PROGRAM PRG_11_AirFlowAnalytics
VAR
	AirFlowRateSensor: GenericSensor;
	AirPressureSensor: GenericSensor;
	AirTemperatureSensor: GenericSensor;
	
	AirFlowSensorPublishMqtt: PublishJsonMqtt;
	AirPresSensorPublishMqtt: PublishJsonMqtt;
	AirTempSensorPublishMqtt: PublishJsonMqtt;
END_VAR

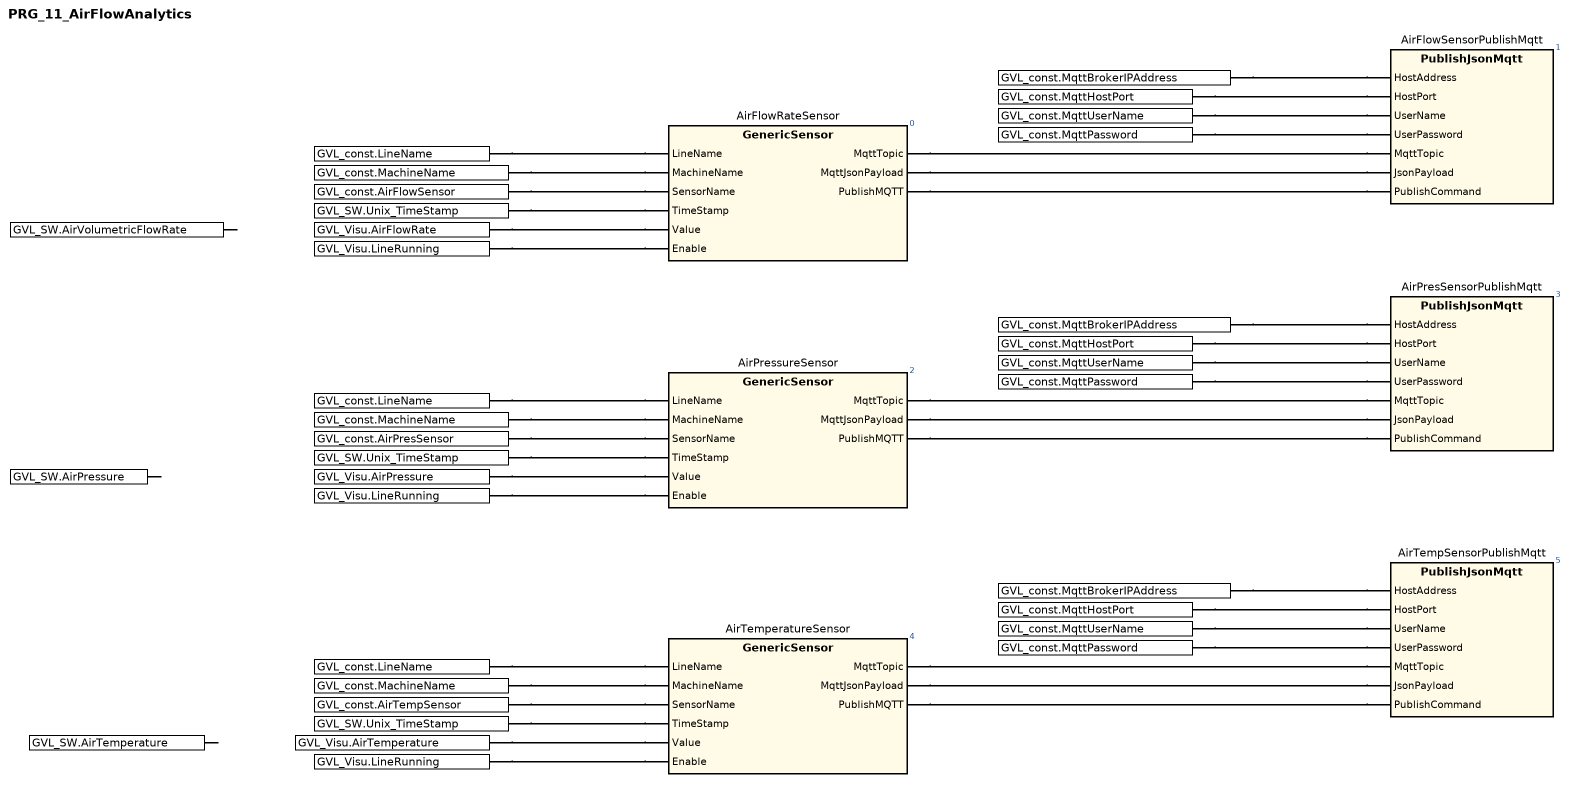
AirFlowRateSensor(
    LineName := GVL_const.LineName,
    MachineName := GVL_const.MachineName,
    SensorName := GVL_const.AirFlowSensor,
    TimeStamp := GVL_SW.Unix_TimeStamp,
    Value := GVL_Visu.AirFlowRate,
    Enable := GVL_Visu.LineRunning); // GenericSensor
AirFlowSensorPublishMqtt(
    HostAddress := GVL_const.MqttBrokerIPAddress,
    HostPort := GVL_const.MqttHostPort,
    UserName := GVL_const.MqttUserName,
    UserPassword := GVL_const.MqttPassword,
    MqttTopic := AirFlowRateSensor.MqttTopic,
    JsonPayload := AirFlowRateSensor.MqttJsonPayload,
    PublishCommand := AirFlowRateSensor.PublishMQTT); // PublishJsonMqtt
AirPressureSensor(
    LineName := GVL_const.LineName,
    MachineName := GVL_const.MachineName,
    SensorName := GVL_const.AirPresSensor,
    TimeStamp := GVL_SW.Unix_TimeStamp,
    Value := GVL_Visu.AirPressure,
    Enable := GVL_Visu.LineRunning); // GenericSensor
AirPresSensorPublishMqtt(
    HostAddress := GVL_const.MqttBrokerIPAddress,
    HostPort := GVL_const.MqttHostPort,
    UserName := GVL_const.MqttUserName,
    UserPassword := GVL_const.MqttPassword,
    MqttTopic := AirPressureSensor.MqttTopic,
    JsonPayload := AirPressureSensor.MqttJsonPayload,
    PublishCommand := AirPressureSensor.PublishMQTT); // PublishJsonMqtt
AirTemperatureSensor(
    LineName := GVL_const.LineName,
    MachineName := GVL_const.MachineName,
    SensorName := GVL_const.AirTempSensor,
    TimeStamp := GVL_SW.Unix_TimeStamp,
    Value := GVL_Visu.AirTemperature,
    Enable := GVL_Visu.LineRunning); // GenericSensor
AirTempSensorPublishMqtt(
    HostAddress := GVL_const.MqttBrokerIPAddress,
    HostPort := GVL_const.MqttHostPort,
    UserName := GVL_const.MqttUserName,
    UserPassword := GVL_const.MqttPassword,
    MqttTopic := AirTemperatureSensor.MqttTopic,
    JsonPayload := AirTemperatureSensor.MqttJsonPayload,
    PublishCommand := AirTemperatureSensor.PublishMQTT); // PublishJsonMqtt
// GVL_SW.AirVolumetricFlowRate: input not connected
// GVL_SW.AirPressure: input not connected
// GVL_SW.AirTemperature: input not connected

END_PROGRAM

(* stored: Version 1.1.0.1, ProductVersion 3.1.4024.15
   POU PRG_11_AirFlowAnalytics: Id {96d35d53-1242-4be7-b36c-7cd64f603641}, SpecialFunc None *)
